INTERFACE GpMotor

METHOD Start : BOOL
VAR_INPUT
END_VAR
END_METHOD

METHOD Stop : BOOL
VAR_INPUT
END_VAR
END_METHOD

END_INTERFACE

(* stored: Version 1.1.0.1, ProductVersion 3.1.4024.16
   Itf GpMotor: Id {ff8d6bf2-a87f-4325-9e3d-a1de3cc13fa5}
   Method Start: Id {93aa7bf5-a726-4e1a-a7e8-bc8b109babab}
   Method Stop: Id {4c84ac34-4de8-4fc5-b5e2-902ab3525fb3} *)
